TYPE ST_AxisAlarm :
STRUCT
    bError       : BOOL;//轴总错误
    nErrorID     : UDINT;//当前优先级最高的错误码
    eErrorSource : E_AxisErrorSource;//错误来源

    bWarning     : BOOL;//警告标志
    nWarningID   : UDINT;//警告码

    eRejectReason : E_AxisRejectReason;//命令拒绝原因
END_STRUCT
END_TYPE

(* stored: Version 1.1.0.1, ProductVersion 3.1.4026.18
   DUT ST_AxisAlarm: Id {026c1a49-80b2-4404-8728-874d0f9ae498} *)
